FUNCTION F_UpdateTimestamp
VAR_INPUT
	stEvents : REFERENCE TO ST_Events;
END_VAR
VAR
	fbGetSystemTime : GETSYSTEMTIME;
	stFileTime : T_FILETIME;
END_VAR


fbGetSystemTime(timeHiDW => stFileTime.dwHighDateTime,
				timeLoDW => stFileTime.dwLowDateTime);

	
stEvents.dtTimestamp := FILETIME_TO_DT (stFileTime);

END_FUNCTION

(* stored: Version 1.1.0.1, ProductVersion 3.1.4024.11
   POU F_UpdateTimestamp: Id {73eb0e1a-3757-4acb-8f61-cd7ad9cad5d8}, SpecialFunc None *)
